// TIA Portal project "thapPhanToNhiPhan" (V14)

(* hardware
DEVICE "S7-1200 station_1"  S7-1200 Station
   slot 0: "Rack_0"  S7-1200 Rack  Rack  V1.0
   slot 1: "PLC_1"  CPU 1214C DC/DC/DC  6ES7 214-1AG40-0XB0  V4.2
*)

// ===== PLC "PLC_1"  CPU 1214C DC/DC/DC =====

VAR_GLOBAL   // PLC tag table "Default tag table"
   "Tag_1" AT %Q0.3 : Bool;
   "Tag_2" AT %I0.0 : Bool;
   "Tag_3" AT %I0.1 : Bool;
   "Tag_4" AT %I0.2 : Bool;
   "Tag_5" AT %I0.3 : Bool;
   "Tag_6" AT %I0.4 : Bool;
   "Tag_7" AT %I0.5 : Bool;
   "Tag_8" AT %I0.6 : Bool;
   "Tag_9" AT %I0.7 : Bool;
END_VAR

ORGANIZATION_BLOCK "Main"   // OB1, LAD, ProgramCycle
TITLE = "Main Program Sweep (Cycle)"
{ S7_Optimized_Access := 'TRUE' }
VERSION : 0.1
   VAR_INPUT
      Initial_Call : Bool;   // Initial call of this OB
      Remanence : Bool;   // =True, if remanent data are available
   END_VAR
BEGIN

REGION Network 1
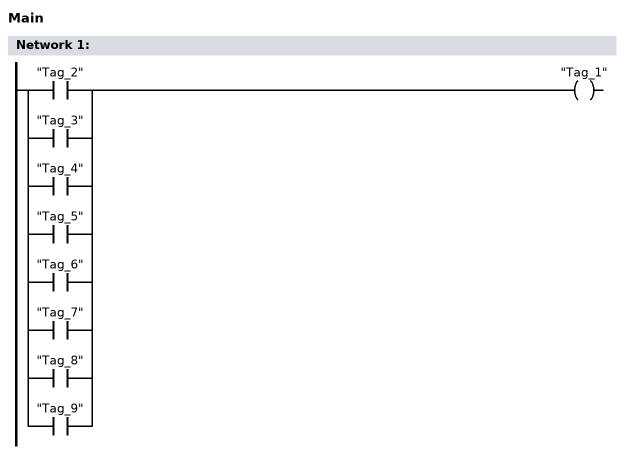
   RUNG wire#powerrail
      Contact( "Tag_2" )
      wire#w1
      Coil( "Tag_1" )
   END_RUNG
   RUNG wire#powerrail
      Contact( "Tag_3" )
   END_RUNG wire#w1
   RUNG wire#powerrail
      Contact( "Tag_4" )
   END_RUNG wire#w1
   RUNG wire#powerrail
      Contact( "Tag_5" )
   END_RUNG wire#w1
   RUNG wire#powerrail
      Contact( "Tag_6" )
   END_RUNG wire#w1
   RUNG wire#powerrail
      Contact( "Tag_7" )
   END_RUNG wire#w1
   RUNG wire#powerrail
      Contact( "Tag_8" )
   END_RUNG wire#w1
   RUNG wire#powerrail
      Contact( "Tag_9" )
   END_RUNG wire#w1
   // the same network as SCL:
   "Tag_1" := "Tag_2" OR "Tag_3" OR "Tag_4" OR "Tag_5" OR "Tag_6" OR "Tag_7" OR "Tag_8" OR "Tag_9";
END_REGION
END_ORGANIZATION_BLOCK